Staubli VAL3: decWriSingIOMsg.pgx

public program decWriSingIOMsg(bool& x_bFlag)
  local num l_nData
  local num l_nIndex
  local num l_nRetVal
begin
  // Copyright (c) 2021, Institute for Factory Automation and Production Systems (FAPS)
  //
  // Licensed under the Apache License, Version 2.0 (the "License");
  // you may not use this file except in compliance with the License.
  // You may obtain a copy of the License at
  //
  //     http://www.apache.org/licenses/LICENSE-2.0
  //
  // Unless required by applicable law or agreed to in writing, software
  // distributed under the License is distributed on an "AS IS" BASIS,
  // WITHOUT WARRANTIES OR CONDITIONS OF ANY KIND, either express or implied.
  // See the License for the specific language governing permissions and
  // limitations under the License.


  // decode write single IO message body (data)

  // assume failure to decode
  writeSingIOMsg.header.nReplyCode=SimpleMsg:ReplyCode.FAILURE

  // fields:
  //  writeSingIOMsg.writeSingleIO.nModuleId
  //  writeSingIOMsg.writeSingleIO.nPin
  //  writeSingIOMsg.writeSingleIO.bState


  // module id, 4 bytes
  l_nRetVal=fromBinary(writeSingIOMsg.body.nData,1,"-4l",writeSingIOMsg.writeSingleIO.nModuleId)
  logMsg(toString("", writeSingIOMsg.body.nData))
  logMsg(toString("", writeSingIOMsg.writeSingleIO.nModuleId))
  logMsg("ID")
  logMsg(toString("", l_nRetVal))
  if(l_nRetVal!=1)
    x_bFlag=false
    return
  endIf

  // pin, 4 bytes
  l_nRetVal=fromBinary(writeSingIOMsg.body.nData[4],1,"-4l",writeSingIOMsg.writeSingleIO.nPin)
  logMsg("pin")
  logMsg(toString("", l_nRetVal))
  if (l_nRetVal!=1)
    x_bFlag=false
    return
  endIf

  // state, 1 byte
  l_nRetVal=fromBinary(writeSingIOMsg.body.nData[8],1,"1",l_nData)
  logMsg("state")
  logMsg(toString("", l_nRetVal))
  if (l_nRetVal!=1)
    x_bFlag=false
    return
  endIf

  // convert decoded data to bool
  if (l_nData==1)
    writeSingIOMsg.writeSingleIO.bState=true
  elseIf (l_nData==0)
    writeSingIOMsg.writeSingleIO.bState=false
  else
    logMsg("[ERROR] WriteSingleIO.bState was decoded to: "+toString("",l_nData))
    x_bFlag=false
    return
  endIf

  // decoding successful
  writeSingIOAck.header.nReplyCode=SimpleMsg:ReplyCode.SUCCESS
  logMsg("SUCCESS")
  x_bFlag=true
end
